{attribute 'GeneratedUsingTerminal: EK1100-0000-0018'}
{attribute addProperty BoxType "EK1100-0000-0018"}
{attribute addProperty Id "Beckhoff_EL30xxEK1122Beckhoff_EL30xxEK1122_6D8563B72A_0001_EL3001_0000_0016EL3001_6939453A21A_0002_EL3001_0000_0017EL3001_353F32DF21A_0003_EL3001_0000_0018EL3001_353F32DF21A_0004_EL3001_0000_0019EL3001_353F32DF21A_0005_EL3001_0000_0020EL3001_353F32DF21A_0006_EL3001_0000_0021EL3001_353F32DF21A_0007_EL3002_0000_0016EL3002_FF9B4B0430A_0008_EL3002_0000_0017EL3002_63BCF66030A_0009_EL3002_0000_0018EL3002_63BCF66030A_0010_EL3002_0000_0019EL3002_63BCF66030A_0011_EL3002_0000_0020EL3002_63BCF66030A_0012_EL3002_0000_0021EL3002_63BCF66030A_0013_EL3004_0000_0016EL3004_E8149C1F48A_0014_EL3004_0000_0017EL3004_C4269E3248A_0015_EL3004_0000_0018EL3004_C4269E3248A_0016_EL3004_0000_0019EL3004_C4269E3248A_0017_EL3004_0000_0020EL3004_C4269E3248A_0018_EL3004_0000_0021EL3004_C4269E3248A_0019_EL3008_0000_0016EL3008_E17B118E84A_0020_EL3008_0000_0017EL3008_335F857B84A_0021_EL3008_0000_0018EL3008_335F857B84A_0022_EL3008_0000_0019EL3008_335F857B84A_0023_EL3008_0000_0020EL3008_335F857B84A_0024_EL3008_0000_0021EL3008_335F857B84A_0025_EL3011_0000_0016EL3011_353F32DF21A_0026_EL3011_0000_0017EL3011_353F32DF21A_0027_EL3011_0000_0018EL3011_353F32DF21A_0028_EL3011_0000_0019EL3011_353F32DF21A_0029_EL3011_0000_0020EL3011_353F32DF21A_0030_EL3012_0000_0016EL3012_63BCF66030A_0031_EL3012_0000_0017EL3012_63BCF66030A_0032_EL3012_0000_0018EL3012_63BCF66030A_0033_EL3012_0000_0019EL3012_63BCF66030A_0034_EL3012_0000_0020EL3012_63BCF66030A_0035_EL3014_0000_0016EL3014_C4269E3248A_0036_EL3014_0000_0017EL3014_C4269E3248A_0037_EL3014_0000_0018EL3014_C4269E3248A_0038_EL3014_0000_0019EL3014_C4269E3248A_0039_EL3021_0000_0016EL3021_353F32DF21A_0040_EL3021_0000_0017EL3021_353F32DF21A_0041_EL3021_0000_0018EL3021_353F32DF21A_0042_EL3021_0000_0019EL3021_353F32DF21A_0043_EL3021_0000_0020EL3021_353F32DF21A_0044_EL3022_0000_0016EL3022_63BCF66030A_0045_EL3022_0000_0017EL3022_63BCF66030A_0046_EL3022_0000_0018EL3022_63BCF66030A_0047_EL3022_0000_0019EL3022_63BCF66030A_0048_EL3022_0000_0020EL3022_63BCF66030A_0049_EL3024_0000_0016EL3024_C4269E3248A_0050_EL3024_0000_0017EL3024_C4269E3248A_0051_EL3024_0000_0018EL3024_C4269E3248A_0052_EL3024_0000_0019EL3024_C4269E3248A_0053_EL3041_0000_0016EL3041_6939453A21A_0054_EL3041_0000_0017EL3041_353F32DF21A_0055_EL3041_0000_0018EL3041_353F32DF21A_0056_EL3041_0000_0019EL3041_353F32DF21A_0057_EL3041_0000_0020EL3041_353F32DF21A_0058_EL3042_0000_0016EL3042_FF9B4B0430A_0059_EL3042_0000_0017EL3042_63BCF66030A_0060_EL3042_0000_0018EL3042_63BCF66030A_0061_EL3042_0000_0019EL3042_63BCF66030A_0062_EL3042_0000_0020EL3042_63BCF66030A_0063_EL3042_0017_0016EL3042_FF9B4B0430A_0064_EL3042_0017_0017EL3042_63BCF66030A_0065_EL3042_0017_0018EL3042_63BCF66030A_0066_EL3042_0017_0019EL3042_63BCF66030A_0067_EL3042_0017_0020EL3042_63BCF66030A_0068_EL3042_0017_0021EL3042_63BCF66030A_0069_EL3044_0000_0016EL3044_E8149C1F48A_0070_EL3044_0000_0017EL3044_C4269E3248A_0071_EL3044_0000_0018EL3044_C4269E3248A_0072_EL3044_0000_0019EL3044_C4269E3248A_0073_EL3044_0000_0020EL3044_C4269E3248A_0074_EL3048_0000_0016EL3048_E17B118E84A_0075_EL3048_0000_0017EL3048_335F857B84A_0076_EL3048_0000_0018EL3048_335F857B84A_0077_EL3048_0000_0019EL3048_335F857B84A_0078_EL3048_0000_0020EL3048_335F857B84A_0079_EL3051_0000_0016EL3051_6939453A21A_0080_EL3051_0000_0017EL3051_353F32DF21A_0081_EL3051_0000_0018EL3051_353F32DF21A_0082_EL3051_0000_0019EL3051_353F32DF21A_0083_EL3051_0000_0020EL3051_353F32DF21A_0084_EL3052_0000_0016EL3052_FF9B4B0430A_0085_EL3052_0000_0017EL3052_63BCF66030A_0086_EL3052_0000_0018EL3052_63BCF66030A_0087_EL3052_0000_0019EL3052_63BCF66030A_0088_EL3052_0000_0020EL3052_63BCF66030A_0089_EL3054_0000_0016EL3054_E8149C1F48A_0090_EL3054_0000_0017EL3054_C4269E3248A_0091_EL3054_0000_0018EL3054_C4269E3248A_0092_EL3054_0000_0019EL3054_C4269E3248A_0093_EL3054_0000_0020EL3054_C4269E3248A_0094_EL3058_0000_0016EL3058_E17B118E84A_0095_EL3058_0000_0017EL3058_335F857B84A_0096_EL3058_0000_0018EL3058_335F857B84A_0097_EL3058_0000_0019EL3058_335F857B84A_0098_EL3058_0000_0020EL3058_335F857B84A_0099_EL3061_0000_0016EL3061_6939453A21A_0100_EL3061_0000_0017EL3061_353F32DF21A_0101_EL3061_0000_0018EL3061_353F32DF21A_0102_EL3061_0000_0019EL3061_353F32DF21A_0103_EL3061_0000_0020EL3061_353F32DF21A_0104_EL3062_0000_0016EL3062_FF9B4B0430A_0105_EL3062_0000_0017EL3062_63BCF66030A_0106_EL3062_0000_0018EL3062_63BCF66030A_0107_EL3062_0000_0019EL3062_63BCF66030A_0108_EL3062_0000_0020EL3062_63BCF66030A_0109_EL3062_0015_0016EL3062_63BCF66030A_0110_EL3062_0030_0016EL3062_FF9B4B0430A_0111_EL3062_0030_0017EL3062_63BCF66030A_0112_EL3062_0030_0018EL3062_63BCF66030A_0113_EL3062_0030_0019EL3062_63BCF66030A_0114_EL3062_0030_0020EL3062_63BCF66030A_0115_EL3062_0030_0021EL3062_63BCF66030A_0116_EL3064_0000_0016EL3064_E8149C1F48A_0117_EL3064_0000_0017EL3064_C4269E3248A_0118_EL3064_0000_0018EL3064_C4269E3248A_0119_EL3064_0000_0019EL3064_C4269E3248A_0120_EL3064_0000_0020EL3064_C4269E3248A_0121_EL3068_0000_0016EL3068_E17B118E84A_0122_EL3068_0000_0017EL3068_335F857B84A_0123_EL3068_0000_0018EL3068_335F857B84A_0124_EL3068_0000_0019EL3068_335F857B84A_0125_EL3068_0000_0020EL3068_335F857B84"}
{attribute addProperty CRC "3588725520"}
{attribute addProperty Size "5129"}
TYPE Beckhoff_EL30xx_D5E79B10 EXTENDS EK1100_1FC0878B :
STRUCT
	{attribute addProperty Name "Beckhoff_EL30xxEK1122"}
	{attribute addProperty PreviousPort "Beckhoff EL30xx : B"}
	Beckhoff_EL30xxEK1122 : Beckhoff_EL30xxEK1122_6D8563B7;
	{attribute addProperty Name "A_0001_EL3001_0000_0016"}
	{attribute addProperty PreviousPort "Beckhoff EL30xxEK1122 : C"}
	A_0001_EL3001_0000_0016 : EL3001_6939453A;
	{attribute addProperty Name "A_0002_EL3001_0000_0017"}
	{attribute addProperty PreviousPort "A_0001(EL3001-0000-0016) : B"}
	A_0002_EL3001_0000_0017 : EL3001_353F32DF;
	{attribute addProperty Name "A_0003_EL3001_0000_0018"}
	{attribute addProperty PreviousPort "A_0002(EL3001-0000-0017) : B"}
	A_0003_EL3001_0000_0018 : EL3001_353F32DF;
	{attribute addProperty Name "A_0004_EL3001_0000_0019"}
	{attribute addProperty PreviousPort "A_0003(EL3001-0000-0018) : B"}
	A_0004_EL3001_0000_0019 : EL3001_353F32DF;
	{attribute addProperty Name "A_0005_EL3001_0000_0020"}
	{attribute addProperty PreviousPort "A_0004(EL3001-0000-0019) : B"}
	A_0005_EL3001_0000_0020 : EL3001_353F32DF;
	{attribute addProperty Name "A_0006_EL3001_0000_0021"}
	{attribute addProperty PreviousPort "A_0005(EL3001-0000-0020) : B"}
	A_0006_EL3001_0000_0021 : EL3001_353F32DF;
	{attribute addProperty Name "A_0007_EL3002_0000_0016"}
	{attribute addProperty PreviousPort "A_0006(EL3001-0000-0021) : B"}
	A_0007_EL3002_0000_0016 : EL3002_FF9B4B04;
	{attribute addProperty Name "A_0008_EL3002_0000_0017"}
	{attribute addProperty PreviousPort "A_0007(EL3002-0000-0016) : B"}
	A_0008_EL3002_0000_0017 : EL3002_63BCF660;
	{attribute addProperty Name "A_0009_EL3002_0000_0018"}
	{attribute addProperty PreviousPort "A_0008(EL3002-0000-0017) : B"}
	A_0009_EL3002_0000_0018 : EL3002_63BCF660;
	{attribute addProperty Name "A_0010_EL3002_0000_0019"}
	{attribute addProperty PreviousPort "A_0009(EL3002-0000-0018) : B"}
	A_0010_EL3002_0000_0019 : EL3002_63BCF660;
	{attribute addProperty Name "A_0011_EL3002_0000_0020"}
	{attribute addProperty PreviousPort "A_0010(EL3002-0000-0019) : B"}
	A_0011_EL3002_0000_0020 : EL3002_63BCF660;
	{attribute addProperty Name "A_0012_EL3002_0000_0021"}
	{attribute addProperty PreviousPort "A_0011(EL3002-0000-0020) : B"}
	A_0012_EL3002_0000_0021 : EL3002_63BCF660;
	{attribute addProperty Name "A_0013_EL3004_0000_0016"}
	{attribute addProperty PreviousPort "A_0012(EL3002-0000-0021) : B"}
	A_0013_EL3004_0000_0016 : EL3004_E8149C1F;
	{attribute addProperty Name "A_0014_EL3004_0000_0017"}
	{attribute addProperty PreviousPort "A_0013(EL3004-0000-0016) : B"}
	A_0014_EL3004_0000_0017 : EL3004_C4269E32;
	{attribute addProperty Name "A_0015_EL3004_0000_0018"}
	{attribute addProperty PreviousPort "A_0014(EL3004-0000-0017) : B"}
	A_0015_EL3004_0000_0018 : EL3004_C4269E32;
	{attribute addProperty Name "A_0016_EL3004_0000_0019"}
	{attribute addProperty PreviousPort "A_0015(EL3004-0000-0018) : B"}
	A_0016_EL3004_0000_0019 : EL3004_C4269E32;
	{attribute addProperty Name "A_0017_EL3004_0000_0020"}
	{attribute addProperty PreviousPort "A_0016(EL3004-0000-0019) : B"}
	A_0017_EL3004_0000_0020 : EL3004_C4269E32;
	{attribute addProperty Name "A_0018_EL3004_0000_0021"}
	{attribute addProperty PreviousPort "A_0017(EL3004-0000-0020) : B"}
	A_0018_EL3004_0000_0021 : EL3004_C4269E32;
	{attribute addProperty Name "A_0019_EL3008_0000_0016"}
	{attribute addProperty PreviousPort "A_0018(EL3004-0000-0021) : B"}
	A_0019_EL3008_0000_0016 : EL3008_E17B118E;
	{attribute addProperty Name "A_0020_EL3008_0000_0017"}
	{attribute addProperty PreviousPort "A_0019(EL3008-0000-0016) : B"}
	A_0020_EL3008_0000_0017 : EL3008_335F857B;
	{attribute addProperty Name "A_0021_EL3008_0000_0018"}
	{attribute addProperty PreviousPort "A_0020(EL3008-0000-0017) : B"}
	A_0021_EL3008_0000_0018 : EL3008_335F857B;
	{attribute addProperty Name "A_0022_EL3008_0000_0019"}
	{attribute addProperty PreviousPort "A_0021(EL3008-0000-0018) : B"}
	A_0022_EL3008_0000_0019 : EL3008_335F857B;
	{attribute addProperty Name "A_0023_EL3008_0000_0020"}
	{attribute addProperty PreviousPort "A_0022(EL3008-0000-0019) : B"}
	A_0023_EL3008_0000_0020 : EL3008_335F857B;
	{attribute addProperty Name "A_0024_EL3008_0000_0021"}
	{attribute addProperty PreviousPort "A_0023(EL3008-0000-0020) : B"}
	A_0024_EL3008_0000_0021 : EL3008_335F857B;
	{attribute addProperty Name "A_0025_EL3011_0000_0016"}
	{attribute addProperty PreviousPort "A_0024(EL3008-0000-0021) : B"}
	A_0025_EL3011_0000_0016 : EL3011_353F32DF;
	{attribute addProperty Name "A_0026_EL3011_0000_0017"}
	{attribute addProperty PreviousPort "A_0025(EL3011-0000-0016) : B"}
	A_0026_EL3011_0000_0017 : EL3011_353F32DF;
	{attribute addProperty Name "A_0027_EL3011_0000_0018"}
	{attribute addProperty PreviousPort "A_0026(EL3011-0000-0017) : B"}
	A_0027_EL3011_0000_0018 : EL3011_353F32DF;
	{attribute addProperty Name "A_0028_EL3011_0000_0019"}
	{attribute addProperty PreviousPort "A_0027(EL3011-0000-0018) : B"}
	A_0028_EL3011_0000_0019 : EL3011_353F32DF;
	{attribute addProperty Name "A_0029_EL3011_0000_0020"}
	{attribute addProperty PreviousPort "A_0028(EL3011-0000-0019) : B"}
	A_0029_EL3011_0000_0020 : EL3011_353F32DF;
	{attribute addProperty Name "A_0030_EL3012_0000_0016"}
	{attribute addProperty PreviousPort "A_0029(EL3011-0000-0020) : B"}
	A_0030_EL3012_0000_0016 : EL3012_63BCF660;
	{attribute addProperty Name "A_0031_EL3012_0000_0017"}
	{attribute addProperty PreviousPort "A_0030(EL3012-0000-0016) : B"}
	A_0031_EL3012_0000_0017 : EL3012_63BCF660;
	{attribute addProperty Name "A_0032_EL3012_0000_0018"}
	{attribute addProperty PreviousPort "A_0031(EL3012-0000-0017) : B"}
	A_0032_EL3012_0000_0018 : EL3012_63BCF660;
	{attribute addProperty Name "A_0033_EL3012_0000_0019"}
	{attribute addProperty PreviousPort "A_0032(EL3012-0000-0018) : B"}
	A_0033_EL3012_0000_0019 : EL3012_63BCF660;
	{attribute addProperty Name "A_0034_EL3012_0000_0020"}
	{attribute addProperty PreviousPort "A_0033(EL3012-0000-0019) : B"}
	A_0034_EL3012_0000_0020 : EL3012_63BCF660;
	{attribute addProperty Name "A_0035_EL3014_0000_0016"}
	{attribute addProperty PreviousPort "A_0034(EL3012-0000-0020) : B"}
	A_0035_EL3014_0000_0016 : EL3014_C4269E32;
	{attribute addProperty Name "A_0036_EL3014_0000_0017"}
	{attribute addProperty PreviousPort "A_0035(EL3014-0000-0016) : B"}
	A_0036_EL3014_0000_0017 : EL3014_C4269E32;
	{attribute addProperty Name "A_0037_EL3014_0000_0018"}
	{attribute addProperty PreviousPort "A_0036(EL3014-0000-0017) : B"}
	A_0037_EL3014_0000_0018 : EL3014_C4269E32;
	{attribute addProperty Name "A_0038_EL3014_0000_0019"}
	{attribute addProperty PreviousPort "A_0037(EL3014-0000-0018) : B"}
	A_0038_EL3014_0000_0019 : EL3014_C4269E32;
	{attribute addProperty Name "A_0039_EL3021_0000_0016"}
	{attribute addProperty PreviousPort "A_0038(EL3014-0000-0019) : B"}
	A_0039_EL3021_0000_0016 : EL3021_353F32DF;
	{attribute addProperty Name "A_0040_EL3021_0000_0017"}
	{attribute addProperty PreviousPort "A_0039(EL3021-0000-0016) : B"}
	A_0040_EL3021_0000_0017 : EL3021_353F32DF;
	{attribute addProperty Name "A_0041_EL3021_0000_0018"}
	{attribute addProperty PreviousPort "A_0040(EL3021-0000-0017) : B"}
	A_0041_EL3021_0000_0018 : EL3021_353F32DF;
	{attribute addProperty Name "A_0042_EL3021_0000_0019"}
	{attribute addProperty PreviousPort "A_0041(EL3021-0000-0018) : B"}
	A_0042_EL3021_0000_0019 : EL3021_353F32DF;
	{attribute addProperty Name "A_0043_EL3021_0000_0020"}
	{attribute addProperty PreviousPort "A_0042(EL3021-0000-0019) : B"}
	A_0043_EL3021_0000_0020 : EL3021_353F32DF;
	{attribute addProperty Name "A_0044_EL3022_0000_0016"}
	{attribute addProperty PreviousPort "A_0043(EL3021-0000-0020) : B"}
	A_0044_EL3022_0000_0016 : EL3022_63BCF660;
	{attribute addProperty Name "A_0045_EL3022_0000_0017"}
	{attribute addProperty PreviousPort "A_0044(EL3022-0000-0016) : B"}
	A_0045_EL3022_0000_0017 : EL3022_63BCF660;
	{attribute addProperty Name "A_0046_EL3022_0000_0018"}
	{attribute addProperty PreviousPort "A_0045(EL3022-0000-0017) : B"}
	A_0046_EL3022_0000_0018 : EL3022_63BCF660;
	{attribute addProperty Name "A_0047_EL3022_0000_0019"}
	{attribute addProperty PreviousPort "A_0046(EL3022-0000-0018) : B"}
	A_0047_EL3022_0000_0019 : EL3022_63BCF660;
	{attribute addProperty Name "A_0048_EL3022_0000_0020"}
	{attribute addProperty PreviousPort "A_0047(EL3022-0000-0019) : B"}
	A_0048_EL3022_0000_0020 : EL3022_63BCF660;
	{attribute addProperty Name "A_0049_EL3024_0000_0016"}
	{attribute addProperty PreviousPort "A_0048(EL3022-0000-0020) : B"}
	A_0049_EL3024_0000_0016 : EL3024_C4269E32;
	{attribute addProperty Name "A_0050_EL3024_0000_0017"}
	{attribute addProperty PreviousPort "A_0049(EL3024-0000-0016) : B"}
	A_0050_EL3024_0000_0017 : EL3024_C4269E32;
	{attribute addProperty Name "A_0051_EL3024_0000_0018"}
	{attribute addProperty PreviousPort "A_0050(EL3024-0000-0017) : B"}
	A_0051_EL3024_0000_0018 : EL3024_C4269E32;
	{attribute addProperty Name "A_0052_EL3024_0000_0019"}
	{attribute addProperty PreviousPort "A_0051(EL3024-0000-0018) : B"}
	A_0052_EL3024_0000_0019 : EL3024_C4269E32;
	{attribute addProperty Name "A_0053_EL3041_0000_0016"}
	{attribute addProperty PreviousPort "A_0052(EL3024-0000-0019) : B"}
	A_0053_EL3041_0000_0016 : EL3041_6939453A;
	{attribute addProperty Name "A_0054_EL3041_0000_0017"}
	{attribute addProperty PreviousPort "A_0053(EL3041-0000-0016) : B"}
	A_0054_EL3041_0000_0017 : EL3041_353F32DF;
	{attribute addProperty Name "A_0055_EL3041_0000_0018"}
	{attribute addProperty PreviousPort "A_0054(EL3041-0000-0017) : B"}
	A_0055_EL3041_0000_0018 : EL3041_353F32DF;
	{attribute addProperty Name "A_0056_EL3041_0000_0019"}
	{attribute addProperty PreviousPort "A_0055(EL3041-0000-0018) : B"}
	A_0056_EL3041_0000_0019 : EL3041_353F32DF;
	{attribute addProperty Name "A_0057_EL3041_0000_0020"}
	{attribute addProperty PreviousPort "A_0056(EL3041-0000-0019) : B"}
	A_0057_EL3041_0000_0020 : EL3041_353F32DF;
	{attribute addProperty Name "A_0058_EL3042_0000_0016"}
	{attribute addProperty PreviousPort "A_0057(EL3041-0000-0020) : B"}
	A_0058_EL3042_0000_0016 : EL3042_FF9B4B04;
	{attribute addProperty Name "A_0059_EL3042_0000_0017"}
	{attribute addProperty PreviousPort "A_0058(EL3042-0000-0016) : B"}
	A_0059_EL3042_0000_0017 : EL3042_63BCF660;
	{attribute addProperty Name "A_0060_EL3042_0000_0018"}
	{attribute addProperty PreviousPort "A_0059(EL3042-0000-0017) : B"}
	A_0060_EL3042_0000_0018 : EL3042_63BCF660;
	{attribute addProperty Name "A_0061_EL3042_0000_0019"}
	{attribute addProperty PreviousPort "A_0060(EL3042-0000-0018) : B"}
	A_0061_EL3042_0000_0019 : EL3042_63BCF660;
	{attribute addProperty Name "A_0062_EL3042_0000_0020"}
	{attribute addProperty PreviousPort "A_0061(EL3042-0000-0019) : B"}
	A_0062_EL3042_0000_0020 : EL3042_63BCF660;
	{attribute addProperty Name "A_0063_EL3042_0017_0016"}
	{attribute addProperty PreviousPort "A_0062(EL3042-0000-0020) : B"}
	A_0063_EL3042_0017_0016 : EL3042_FF9B4B04;
	{attribute addProperty Name "A_0064_EL3042_0017_0017"}
	{attribute addProperty PreviousPort "A_0063(EL3042-0017-0016) : B"}
	A_0064_EL3042_0017_0017 : EL3042_63BCF660;
	{attribute addProperty Name "A_0065_EL3042_0017_0018"}
	{attribute addProperty PreviousPort "A_0064(EL3042-0017-0017) : B"}
	A_0065_EL3042_0017_0018 : EL3042_63BCF660;
	{attribute addProperty Name "A_0066_EL3042_0017_0019"}
	{attribute addProperty PreviousPort "A_0065(EL3042-0017-0018) : B"}
	A_0066_EL3042_0017_0019 : EL3042_63BCF660;
	{attribute addProperty Name "A_0067_EL3042_0017_0020"}
	{attribute addProperty PreviousPort "A_0066(EL3042-0017-0019) : B"}
	A_0067_EL3042_0017_0020 : EL3042_63BCF660;
	{attribute addProperty Name "A_0068_EL3042_0017_0021"}
	{attribute addProperty PreviousPort "A_0067(EL3042-0017-0020) : B"}
	A_0068_EL3042_0017_0021 : EL3042_63BCF660;
	{attribute addProperty Name "A_0069_EL3044_0000_0016"}
	{attribute addProperty PreviousPort "A_0068(EL3042-0017-0021) : B"}
	A_0069_EL3044_0000_0016 : EL3044_E8149C1F;
	{attribute addProperty Name "A_0070_EL3044_0000_0017"}
	{attribute addProperty PreviousPort "A_0069(EL3044-0000-0016) : B"}
	A_0070_EL3044_0000_0017 : EL3044_C4269E32;
	{attribute addProperty Name "A_0071_EL3044_0000_0018"}
	{attribute addProperty PreviousPort "A_0070(EL3044-0000-0017) : B"}
	A_0071_EL3044_0000_0018 : EL3044_C4269E32;
	{attribute addProperty Name "A_0072_EL3044_0000_0019"}
	{attribute addProperty PreviousPort "A_0071(EL3044-0000-0018) : B"}
	A_0072_EL3044_0000_0019 : EL3044_C4269E32;
	{attribute addProperty Name "A_0073_EL3044_0000_0020"}
	{attribute addProperty PreviousPort "A_0072(EL3044-0000-0019) : B"}
	A_0073_EL3044_0000_0020 : EL3044_C4269E32;
	{attribute addProperty Name "A_0074_EL3048_0000_0016"}
	{attribute addProperty PreviousPort "A_0073(EL3044-0000-0020) : B"}
	A_0074_EL3048_0000_0016 : EL3048_E17B118E;
	{attribute addProperty Name "A_0075_EL3048_0000_0017"}
	{attribute addProperty PreviousPort "A_0074(EL3048-0000-0016) : B"}
	A_0075_EL3048_0000_0017 : EL3048_335F857B;
	{attribute addProperty Name "A_0076_EL3048_0000_0018"}
	{attribute addProperty PreviousPort "A_0075(EL3048-0000-0017) : B"}
	A_0076_EL3048_0000_0018 : EL3048_335F857B;
	{attribute addProperty Name "A_0077_EL3048_0000_0019"}
	{attribute addProperty PreviousPort "A_0076(EL3048-0000-0018) : B"}
	A_0077_EL3048_0000_0019 : EL3048_335F857B;
	{attribute addProperty Name "A_0078_EL3048_0000_0020"}
	{attribute addProperty PreviousPort "A_0077(EL3048-0000-0019) : B"}
	A_0078_EL3048_0000_0020 : EL3048_335F857B;
	{attribute addProperty Name "A_0079_EL3051_0000_0016"}
	{attribute addProperty PreviousPort "A_0078(EL3048-0000-0020) : B"}
	A_0079_EL3051_0000_0016 : EL3051_6939453A;
	{attribute addProperty Name "A_0080_EL3051_0000_0017"}
	{attribute addProperty PreviousPort "A_0079(EL3051-0000-0016) : B"}
	A_0080_EL3051_0000_0017 : EL3051_353F32DF;
	{attribute addProperty Name "A_0081_EL3051_0000_0018"}
	{attribute addProperty PreviousPort "A_0080(EL3051-0000-0017) : B"}
	A_0081_EL3051_0000_0018 : EL3051_353F32DF;
	{attribute addProperty Name "A_0082_EL3051_0000_0019"}
	{attribute addProperty PreviousPort "A_0081(EL3051-0000-0018) : B"}
	A_0082_EL3051_0000_0019 : EL3051_353F32DF;
	{attribute addProperty Name "A_0083_EL3051_0000_0020"}
	{attribute addProperty PreviousPort "A_0082(EL3051-0000-0019) : B"}
	A_0083_EL3051_0000_0020 : EL3051_353F32DF;
	{attribute addProperty Name "A_0084_EL3052_0000_0016"}
	{attribute addProperty PreviousPort "A_0083(EL3051-0000-0020) : B"}
	A_0084_EL3052_0000_0016 : EL3052_FF9B4B04;
	{attribute addProperty Name "A_0085_EL3052_0000_0017"}
	{attribute addProperty PreviousPort "A_0084(EL3052-0000-0016) : B"}
	A_0085_EL3052_0000_0017 : EL3052_63BCF660;
	{attribute addProperty Name "A_0086_EL3052_0000_0018"}
	{attribute addProperty PreviousPort "A_0085(EL3052-0000-0017) : B"}
	A_0086_EL3052_0000_0018 : EL3052_63BCF660;
	{attribute addProperty Name "A_0087_EL3052_0000_0019"}
	{attribute addProperty PreviousPort "A_0086(EL3052-0000-0018) : B"}
	A_0087_EL3052_0000_0019 : EL3052_63BCF660;
	{attribute addProperty Name "A_0088_EL3052_0000_0020"}
	{attribute addProperty PreviousPort "A_0087(EL3052-0000-0019) : B"}
	A_0088_EL3052_0000_0020 : EL3052_63BCF660;
	{attribute addProperty Name "A_0089_EL3054_0000_0016"}
	{attribute addProperty PreviousPort "A_0088(EL3052-0000-0020) : B"}
	A_0089_EL3054_0000_0016 : EL3054_E8149C1F;
	{attribute addProperty Name "A_0090_EL3054_0000_0017"}
	{attribute addProperty PreviousPort "A_0089(EL3054-0000-0016) : B"}
	A_0090_EL3054_0000_0017 : EL3054_C4269E32;
	{attribute addProperty Name "A_0091_EL3054_0000_0018"}
	{attribute addProperty PreviousPort "A_0090(EL3054-0000-0017) : B"}
	A_0091_EL3054_0000_0018 : EL3054_C4269E32;
	{attribute addProperty Name "A_0092_EL3054_0000_0019"}
	{attribute addProperty PreviousPort "A_0091(EL3054-0000-0018) : B"}
	A_0092_EL3054_0000_0019 : EL3054_C4269E32;
	{attribute addProperty Name "A_0093_EL3054_0000_0020"}
	{attribute addProperty PreviousPort "A_0092(EL3054-0000-0019) : B"}
	A_0093_EL3054_0000_0020 : EL3054_C4269E32;
	{attribute addProperty Name "A_0094_EL3058_0000_0016"}
	{attribute addProperty PreviousPort "A_0093(EL3054-0000-0020) : B"}
	A_0094_EL3058_0000_0016 : EL3058_E17B118E;
	{attribute addProperty Name "A_0095_EL3058_0000_0017"}
	{attribute addProperty PreviousPort "A_0094(EL3058-0000-0016) : B"}
	A_0095_EL3058_0000_0017 : EL3058_335F857B;
	{attribute addProperty Name "A_0096_EL3058_0000_0018"}
	{attribute addProperty PreviousPort "A_0095(EL3058-0000-0017) : B"}
	A_0096_EL3058_0000_0018 : EL3058_335F857B;
	{attribute addProperty Name "A_0097_EL3058_0000_0019"}
	{attribute addProperty PreviousPort "A_0096(EL3058-0000-0018) : B"}
	A_0097_EL3058_0000_0019 : EL3058_335F857B;
	{attribute addProperty Name "A_0098_EL3058_0000_0020"}
	{attribute addProperty PreviousPort "A_0097(EL3058-0000-0019) : B"}
	A_0098_EL3058_0000_0020 : EL3058_335F857B;
	{attribute addProperty Name "A_0099_EL3061_0000_0016"}
	{attribute addProperty PreviousPort "A_0098(EL3058-0000-0020) : B"}
	A_0099_EL3061_0000_0016 : EL3061_6939453A;
	{attribute addProperty Name "A_0100_EL3061_0000_0017"}
	{attribute addProperty PreviousPort "A_0099(EL3061-0000-0016) : B"}
	A_0100_EL3061_0000_0017 : EL3061_353F32DF;
	{attribute addProperty Name "A_0101_EL3061_0000_0018"}
	{attribute addProperty PreviousPort "A_0100(EL3061-0000-0017) : B"}
	A_0101_EL3061_0000_0018 : EL3061_353F32DF;
	{attribute addProperty Name "A_0102_EL3061_0000_0019"}
	{attribute addProperty PreviousPort "A_0101(EL3061-0000-0018) : B"}
	A_0102_EL3061_0000_0019 : EL3061_353F32DF;
	{attribute addProperty Name "A_0103_EL3061_0000_0020"}
	{attribute addProperty PreviousPort "A_0102(EL3061-0000-0019) : B"}
	A_0103_EL3061_0000_0020 : EL3061_353F32DF;
	{attribute addProperty Name "A_0104_EL3062_0000_0016"}
	{attribute addProperty PreviousPort "A_0103(EL3061-0000-0020) : B"}
	A_0104_EL3062_0000_0016 : EL3062_FF9B4B04;
	{attribute addProperty Name "A_0105_EL3062_0000_0017"}
	{attribute addProperty PreviousPort "A_0104(EL3062-0000-0016) : B"}
	A_0105_EL3062_0000_0017 : EL3062_63BCF660;
	{attribute addProperty Name "A_0106_EL3062_0000_0018"}
	{attribute addProperty PreviousPort "A_0105(EL3062-0000-0017) : B"}
	A_0106_EL3062_0000_0018 : EL3062_63BCF660;
	{attribute addProperty Name "A_0107_EL3062_0000_0019"}
	{attribute addProperty PreviousPort "A_0106(EL3062-0000-0018) : B"}
	A_0107_EL3062_0000_0019 : EL3062_63BCF660;
	{attribute addProperty Name "A_0108_EL3062_0000_0020"}
	{attribute addProperty PreviousPort "A_0107(EL3062-0000-0019) : B"}
	A_0108_EL3062_0000_0020 : EL3062_63BCF660;
	{attribute addProperty Name "A_0109_EL3062_0015_0016"}
	{attribute addProperty PreviousPort "A_0108(EL3062-0000-0020) : B"}
	A_0109_EL3062_0015_0016 : EL3062_63BCF660;
	{attribute addProperty Name "A_0110_EL3062_0030_0016"}
	{attribute addProperty PreviousPort "A_0109(EL3062-0015-0016) : B"}
	A_0110_EL3062_0030_0016 : EL3062_FF9B4B04;
	{attribute addProperty Name "A_0111_EL3062_0030_0017"}
	{attribute addProperty PreviousPort "A_0110(EL3062-0030-0016) : B"}
	A_0111_EL3062_0030_0017 : EL3062_63BCF660;
	{attribute addProperty Name "A_0112_EL3062_0030_0018"}
	{attribute addProperty PreviousPort "A_0111(EL3062-0030-0017) : B"}
	A_0112_EL3062_0030_0018 : EL3062_63BCF660;
	{attribute addProperty Name "A_0113_EL3062_0030_0019"}
	{attribute addProperty PreviousPort "A_0112(EL3062-0030-0018) : B"}
	A_0113_EL3062_0030_0019 : EL3062_63BCF660;
	{attribute addProperty Name "A_0114_EL3062_0030_0020"}
	{attribute addProperty PreviousPort "A_0113(EL3062-0030-0019) : B"}
	A_0114_EL3062_0030_0020 : EL3062_63BCF660;
	{attribute addProperty Name "A_0115_EL3062_0030_0021"}
	{attribute addProperty PreviousPort "A_0114(EL3062-0030-0020) : B"}
	A_0115_EL3062_0030_0021 : EL3062_63BCF660;
	{attribute addProperty Name "A_0116_EL3064_0000_0016"}
	{attribute addProperty PreviousPort "A_0115(EL3062-0030-0021) : B"}
	A_0116_EL3064_0000_0016 : EL3064_E8149C1F;
	{attribute addProperty Name "A_0117_EL3064_0000_0017"}
	{attribute addProperty PreviousPort "A_0116(EL3064-0000-0016) : B"}
	A_0117_EL3064_0000_0017 : EL3064_C4269E32;
	{attribute addProperty Name "A_0118_EL3064_0000_0018"}
	{attribute addProperty PreviousPort "A_0117(EL3064-0000-0017) : B"}
	A_0118_EL3064_0000_0018 : EL3064_C4269E32;
	{attribute addProperty Name "A_0119_EL3064_0000_0019"}
	{attribute addProperty PreviousPort "A_0118(EL3064-0000-0018) : B"}
	A_0119_EL3064_0000_0019 : EL3064_C4269E32;
	{attribute addProperty Name "A_0120_EL3064_0000_0020"}
	{attribute addProperty PreviousPort "A_0119(EL3064-0000-0019) : B"}
	A_0120_EL3064_0000_0020 : EL3064_C4269E32;
	{attribute addProperty Name "A_0121_EL3068_0000_0016"}
	{attribute addProperty PreviousPort "A_0120(EL3064-0000-0020) : B"}
	A_0121_EL3068_0000_0016 : EL3068_E17B118E;
	{attribute addProperty Name "A_0122_EL3068_0000_0017"}
	{attribute addProperty PreviousPort "A_0121(EL3068-0000-0016) : B"}
	A_0122_EL3068_0000_0017 : EL3068_335F857B;
	{attribute addProperty Name "A_0123_EL3068_0000_0018"}
	{attribute addProperty PreviousPort "A_0122(EL3068-0000-0017) : B"}
	A_0123_EL3068_0000_0018 : EL3068_335F857B;
	{attribute addProperty Name "A_0124_EL3068_0000_0019"}
	{attribute addProperty PreviousPort "A_0123(EL3068-0000-0018) : B"}
	A_0124_EL3068_0000_0019 : EL3068_335F857B;
	{attribute addProperty Name "A_0125_EL3068_0000_0020"}
	{attribute addProperty PreviousPort "A_0124(EL3068-0000-0019) : B"}
	A_0125_EL3068_0000_0020 : EL3068_335F857B;
END_STRUCT
END_TYPE

(* stored: Version 1.2.0.0, ProductVersion 3.1.4024.9
   DUT Beckhoff_EL30xx_D5E79B10: Id {f26fde35-25b8-4ed6-862d-20075580d806} *)
